TYPE ST_ComboboxEntry :
STRUCT    
	id : INT;
    text : STRING;
    value : INT;
END_STRUCT
END_TYPE

(* stored: Version 1.1.0.1
   DUT ST_ComboboxEntry: Id {08af3126-3438-46cc-8175-7bf5eb347fdf} *)
